(* CODESYS project sklep_GK.project

Project tree, tasks and I/O mapping:
  Device : CODESYS Control Win V3, CODESYS, version 3.5.20.30
    application Application
      libraries: Standard, 3.5.18.0 (System); VisuDialogs, * (System)
      task VISU_TASK (cyclic, interval 100 ms, priority 31) calls VisuElems.Visu_Prg
      task MainTask (cyclic, interval t#20ms, priority 1) calls PLC_PRG_GK
      visualisation Visualization
      program PLC_PRG_GK [LD]
  libraries: Standard, 3.5.18.0 (System); VisuElemBase, * (System)
  text list GlobalTextList
*)

// Device/Application/PLC_PRG_GK
PROGRAM PLC_PRG_GK
VAR
    start_GK, zatrzymanie_Pracy_GK:BOOL;
    H1_GK, H2_GK, H3_GK: BOOL;
	M1_GK,M2_GK, M3_GK: BOOL;
 	B1_GK,B2_GK: BOOL;
	LDH2_GK,LGH2_GK,LDH3_GK:WORD;
	liczba_klientow_GK:WORD;
	intruz_GK:BOOL;
	restart_systemu_GK:BOOL;
	
	
	CTUD_GK: CTUD;
END_VAR
VAR // added by the converter: edge detectors and wires of the graphical bodies
    _w1 : BOOL;
END_VAR

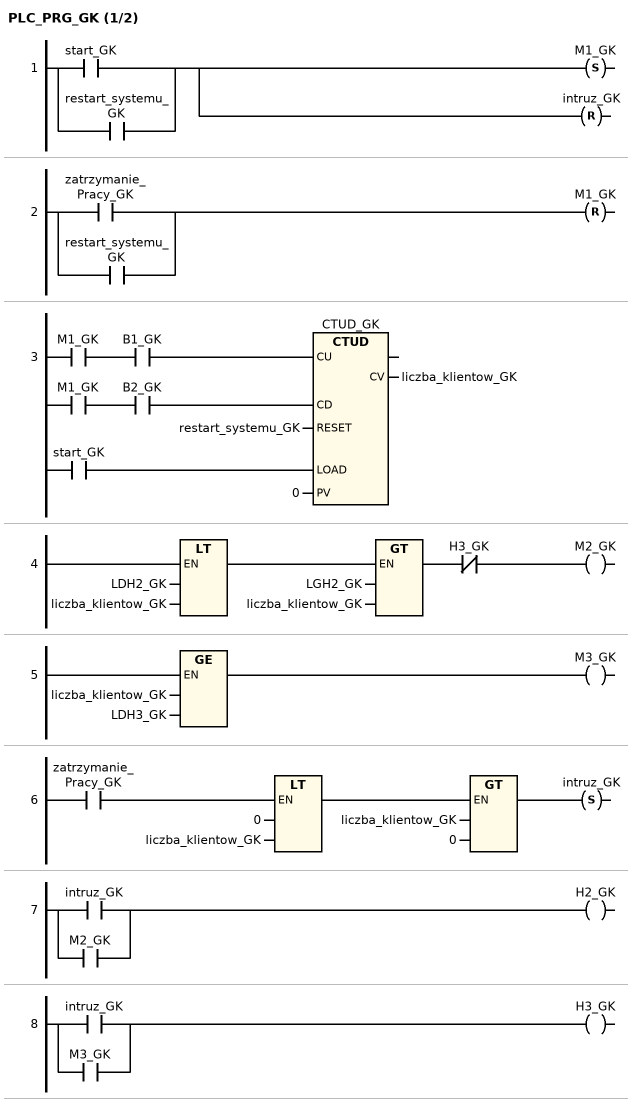
// NETWORK 1
_w1 := start_GK OR restart_systemu_GK;
M1_GK S= _w1;
intruz_GK R= _w1;

// NETWORK 2
M1_GK R= zatrzymanie_Pracy_GK OR restart_systemu_GK;

// NETWORK 3
CTUD_GK(
    CU := M1_GK AND B1_GK,
    CD := M1_GK AND B2_GK,
    RESET := restart_systemu_GK,
    LOAD := start_GK,
    PV := 0,
    CV => liczba_klientow_GK); // CTUD

// NETWORK 4
M2_GK := (LDH2_GK < liczba_klientow_GK AND LGH2_GK > liczba_klientow_GK) AND NOT H3_GK;

// NETWORK 5
M3_GK := liczba_klientow_GK >= LDH3_GK;

// NETWORK 6
intruz_GK S= zatrzymanie_Pracy_GK AND 0 < liczba_klientow_GK AND liczba_klientow_GK > 0;

// NETWORK 7
H2_GK := intruz_GK OR M2_GK;

// NETWORK 8
H3_GK := intruz_GK OR M3_GK;

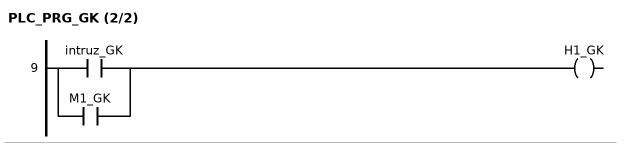
// NETWORK 9
H1_GK := intruz_GK OR M1_GK;

END_PROGRAM

// Device/Application/Visualization
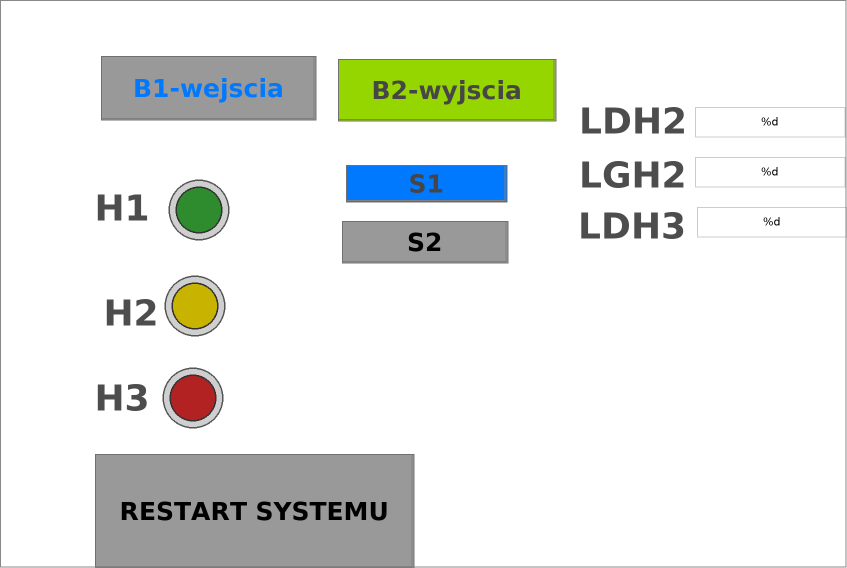
VISUALIZATION Visualization  // 847x568
    Lamp1 (164,175 70x70), variable: PLC_PRG_GK.H1_GK, style: Lamp-Lamp1-Green
    Lamp1 (160,271 70x70), variable: PLC_PRG_GK.H2_GK, style: Lamp-Lamp1-Yellow
    Lamp1 (158,363 70x70), variable: PLC_PRG_GK.H3_GK, style: Lamp-Lamp1-Red
    Button (342,221 166x42), "S2"
        tap PLC_PRG_GK.zatrzymanie_Pracy_GK
    Button (101,56 215x64), "B1-wejscia"
        tap PLC_PRG_GK.B1_GK
    Button (338,59 218x62), "B2-wyjscia"
        tap PLC_PRG_GK.B2_GK
    Button (346,165 161x37), "S1"
        tap PLC_PRG_GK.start_GK
    Label (558,106 150x30), "LDH2"
    Label (47,193 150x30), "H1"
    Label (47,383 150x30), "H3"
    Textfield (695,107 150x30), "%d", text variable: PLC_PRG_GK.LDH2_GK
        OnMouseClick: write the text variable via Default
    Textfield (695,157 150x30), "%d", text variable: PLC_PRG_GK.LGH2_GK
        OnMouseClick: write the text variable via Default
    Textfield (697,207 150x30), "%d", text variable: PLC_PRG_GK.LDH3_GK
        OnMouseClick: write the text variable via Default
    Label (56,298 150x30), "H2"
    Label (557,211 150x30), "LDH3"
    Label (558,160 150x30), "LGH2"
    Button (95,454 319x114), "RESTART SYSTEMU"
        tap PLC_PRG_GK.restart_systemu_GK
END_VISUALIZATION
